TEXTLIST TL_EventType
  0 = ''
  1 = 'Alarm'
  2 = 'Message'
   = ''
END_TEXTLIST

(* stored: Version 1.1.0.1, ProductVersion 3.1.4024.9
   TextList TL_EventType: Id {b6d65e14-2db5-420d-864a-5ae6c615236c} *)
